FUNCTION_BLOCK xaxpy_dm
VAR_INPUT
    b_n: DINT;
    a: LREAL;
    x: ARRAY [0..5] OF LREAL;
    ix0: DINT;
    iy0: DINT;
END_VAR
VAR_IN_OUT
    y: ARRAY [0..29] OF LREAL;
END_VAR
VAR_TEMP
    ix: DINT;
    iy: DINT;
    k: DINT;
END_VAR

IF (b_n >= 1) AND (a <> 0.0) THEN 
    ix := ix0 - 1;
    iy := iy0 - 1;
    k := 0;
    WHILE k <= (b_n - 1) DO
        y[iy] := (a * x[ix]) + y[iy];
        ix := ix + 1;
        iy := iy + 1;
        k := k + 1;
    END_WHILE;
END_IF;

END_FUNCTION_BLOCK

(* stored: Version 1.1.0.1, ProductVersion 3.1.4024.12
   POU xaxpy_dm: Id {5ad1c8f5-e470-41b8-adbb-f2020b51c24b}, SpecialFunc None *)
